// Mitsubishi GX Works2 project: 신호등   PLC: Q03UDV

PROGRAM MAIN
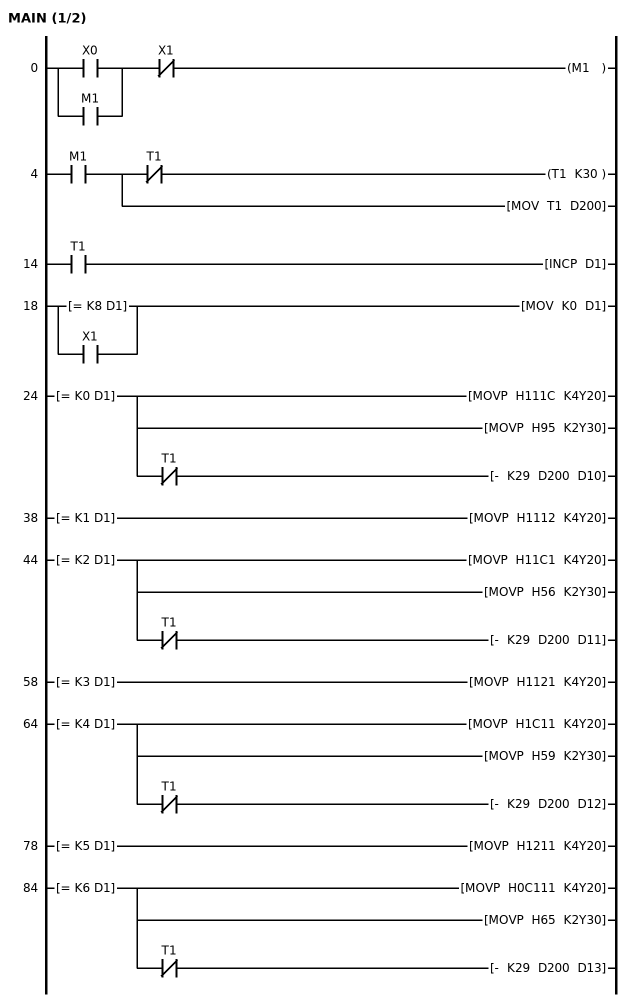
0     LD      X0
      OR      M1
      ANI     X1
      OUT     M1
4     LD      M1
      MPS
      ANI     T1
      OUT     T1 K30
      MPP
      MOV     T1 D200
14    LD      T1
      INCP    D1
18    LD=     K8 D1
      OR      X1
      MOV     K0 D1
24    LD=     K0 D1
      MOVP    H111C K4Y20
      MOVP    H95 K2Y30
      ANI     T1
      -       K29 D200 D10
38    LD=     K1 D1
      MOVP    H1112 K4Y20
44    LD=     K2 D1
      MOVP    H11C1 K4Y20
      MOVP    H56 K2Y30
      ANI     T1
      -       K29 D200 D11
58    LD=     K3 D1
      MOVP    H1121 K4Y20
64    LD=     K4 D1
      MOVP    H1C11 K4Y20
      MOVP    H59 K2Y30
      ANI     T1
      -       K29 D200 D12
78    LD=     K5 D1
      MOVP    H1211 K4Y20
84    LD=     K6 D1
      MOVP    H0C111 K4Y20
      MOVP    H65 K2Y30
      ANI     T1
      -       K29 D200 D13
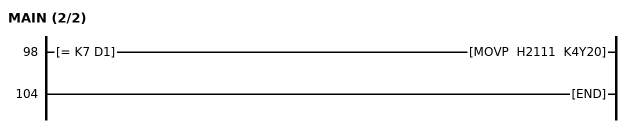
98    LD=     K7 D1
      MOVP    H2111 K4Y20
104   END
END_PROGRAM
